// TIA Portal V20 export
TYPE "CMInterface_DO"
   STRUCT
      Output { ExternalAccessible := 'False'; ExternalVisible := 'False'; ExternalWritable := 'False'} : Bool;
   END_STRUCT;
END_TYPE
